FUNCTION_BLOCK FlushCdt (* CAT Function Block Type *)
  (* Standard: 61499-2 *)
  (* Version 0.0, 6/7/2026, Schneider Electric, template *)
  PACKAGE SE.Nereda;
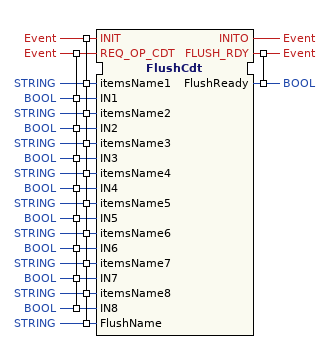
  EVENT_INPUT
    INIT WITH itemsName1, itemsName2, itemsName3, itemsName4, itemsName5, itemsName6, itemsName7, itemsName8, FlushName;
    REQ_OP_CDT WITH IN1, IN2, IN3, IN4, IN5, IN6, IN7, IN8; (* Normal Execution Request *)
  END_EVENT
  EVENT_OUTPUT
    INITO;
    FLUSH_RDY WITH FlushReady; (* Input changed *)
  END_EVENT
  VAR_INPUT
    itemsName1 : STRING;
    IN1 : BOOL; (* Argument *)
    itemsName2 : STRING;
    IN2 : BOOL; (* Argument *)
    itemsName3 : STRING;
    IN3 : BOOL; (* Argument *)
    itemsName4 : STRING;
    IN4 : BOOL; (* Argument *)
    itemsName5 : STRING;
    IN5 : BOOL; (* Argument *)
    itemsName6 : STRING;
    IN6 : BOOL; (* Argument *)
    itemsName7 : STRING;
    IN7 : BOOL; (* Argument *)
    itemsName8 : STRING;
    IN8 : BOOL; (* Argument *)
    FlushName : STRING;
  END_VAR
  VAR_OUTPUT
    FlushReady : BOOL; (* Output value *)
  END_VAR
  (* 01 - FUNCTIONNAL INPUT INTERFACE *)
  (* 05 - LOGIC *)
  (* 02 - FUNCTIONNAL OUTPUT INTERFACE *)
  (* 00 - INITIALIZATION *)
  (* 06 - HMI INTERFACE *)
  (* 03 - FIELD INTERFACE *)
  FBS
    OpCdts : AND_8036BCB1C7C04BD2; {SET_ATTRIBUTE(Configuration.GenericFBType.InterfaceParams, Runtime.Standard#CNT:=8;OUT:BOOL)}
    encodeB1 : VALFORMAT_95B1C22C7F49B890(FORMAT := '%s%s%s%s'); {SET_ATTRIBUTE(Configuration.GenericFBType.InterfaceParams, Runtime.Standard#I:=4;VALUE${I$}:INT,INT,INT,INT)}
    encodeB2 : VALFORMAT_95B1C22C7F49B890(FORMAT := '%s%s%s%s'); {SET_ATTRIBUTE(Configuration.GenericFBType.InterfaceParams, Runtime.Standard#I:=4;VALUE${I$}:INT,INT,INT,INT)}
    OpCdtsSmooth : boolValueChanged;
    IThis : FlushCdt_HMI(QI := TRUE);
    ForceCdts : OR_88A3DD8EC65DD11C; {SET_ATTRIBUTE(Configuration.GenericFBType.InterfaceParams, Runtime.Standard#CNT:=2;OUT:BOOL)}
    STR2INT1 : STR2INT;
    STR2INT2 : STR2INT;
    BOOL2INT1 : BOOL2INT_4;
    BOOL2INT2 : BOOL2INT_4;
  END_FBS
  EVENT_CONNECTIONS
    OpCdtsSmooth.CHD TO FLUSH_RDY;
    REQ_OP_CDT TO OpCdts.REQ;
    OpCdts.CNF TO ForceCdts.REQ;
    ForceCdts.CNF TO OpCdtsSmooth.REQ;
    BOOL2INT1.6FC99A5BD1C38561 TO encodeB1.REQ;
    encodeB1.CNF TO STR2INT1.DD5870AA881150BB;
    BOOL2INT2.6FC99A5BD1C38561 TO encodeB2.REQ;
    encodeB2.CNF TO STR2INT2.DD5870AA881150BB;
    INIT TO IThis.7D98611DC811A4F7;
    OpCdtsSmooth.CNF TO IThis.A7C33F064CCD848C;
    IThis.8A8403C8DB481D6C TO IThis.6D29BCFC45D76FE3;
    IThis.8A8403C8DB481D6C TO IThis.A665539B906F6DBA;
    IThis.8A8403C8DB481D6C TO INITO;
    IThis.740E64ACF018D1C7 TO OpCdts.REQ;
    STR2INT1.6FC99A5BD1C38561 TO BOOL2INT2.DD5870AA881150BB;
    STR2INT2.6FC99A5BD1C38561 TO IThis.6D29BCFC45D76FE3;
    OpCdtsSmooth.CNF TO BOOL2INT1.DD5870AA881150BB;
  END_CONNECTIONS
  DATA_CONNECTIONS
    OpCdtsSmooth.Output TO FlushReady;
    IN1 TO OpCdts.IN1;
    IN2 TO OpCdts.IN2;
    IN3 TO OpCdts.IN3;
    IN4 TO OpCdts.IN4;
    IN5 TO OpCdts.IN5;
    IN6 TO OpCdts.IN6;
    IN7 TO OpCdts.IN7;
    IN8 TO OpCdts.IN8;
    OpCdts.OUT TO ForceCdts.IN1;
    ForceCdts.OUT TO OpCdtsSmooth.Input;
    BOOL2INT1.A6DEF5F9C27C1848 TO encodeB1.VALUE1;
    BOOL2INT1.515A2E3BB78F58C7 TO encodeB1.VALUE2;
    BOOL2INT1.FCA64FB4B13F606F TO encodeB1.VALUE3;
    BOOL2INT1.740A810221DABFBE TO encodeB1.VALUE4;
    encodeB1.RESULT TO STR2INT1.4573FC8F228EB71D;
    BOOL2INT2.A6DEF5F9C27C1848 TO encodeB2.VALUE1;
    BOOL2INT2.515A2E3BB78F58C7 TO encodeB2.VALUE2;
    BOOL2INT2.FCA64FB4B13F606F TO encodeB2.VALUE3;
    BOOL2INT2.740A810221DABFBE TO encodeB2.VALUE4;
    encodeB2.RESULT TO STR2INT2.4573FC8F228EB71D;
    OpCdtsSmooth.Output TO IThis.52F65A7B68D385BC;
    FlushName TO IThis.5F8F361E80D292F1;
    itemsName1 TO IThis.74E1E0951D70046E;
    itemsName2 TO IThis.EE9470BA0350B131;
    itemsName3 TO IThis.EDAEBE4CEBDB9AE9;
    itemsName4 TO IThis.521EB392A39EAFAC;
    itemsName5 TO IThis.882EBDE88CE34770;
    itemsName6 TO IThis.CFFC3D70D2D95759;
    itemsName7 TO IThis.FEED97F6C5CA5C81;
    itemsName8 TO IThis.7E2A6F1CECD5D852;
    STR2INT1.A6DEF5F9C27C1848 TO IThis.9CD6AD33A52FBF26;
    STR2INT2.A6DEF5F9C27C1848 TO IThis.CC812AEED2D2840D;
    IThis.767754EBE4FABC5A TO ForceCdts.IN2;
    IN4 TO BOOL2INT1.4573FC8F228EB71D;
    IN3 TO BOOL2INT1.DF8224FEB3446E92;
    IN2 TO BOOL2INT1.F547CEFAFDE5D422;
    IN1 TO BOOL2INT1.25941BC08BA9FF7D;
    IN8 TO BOOL2INT2.4573FC8F228EB71D;
    IN7 TO BOOL2INT2.DF8224FEB3446E92;
    IN6 TO BOOL2INT2.F547CEFAFDE5D422;
    IN5 TO BOOL2INT2.25941BC08BA9FF7D;
  END_CONNECTIONS
END_FUNCTION_BLOCK
